// TIA Portal V17 export
// export: Created 2025-03-07T09:24:28.1169824Z, ExportSetting WithDefaults, DisplayName Totally Integrated Automation Portal, DisplayVersion V17 Update 8, DisplayName TIA Portal Openness, DisplayVersion V17 Update 8, DisplayName TIA Portal Version Control Interface, DisplayVersion V17, DisplayName SINAMICS Startdrive Advanced, DisplayVersion V17 SP2, DisplayName SINAMICS Startdrive G110M, G120, G120C, G120D, G120P, G115D, DisplayVersion V17 SP2, DisplayName SINAMICS Startdrive G130, G150, S120, S150, SINAMICS MV, S210, DisplayVersion V17 SP2, DisplayName STEP 7 Professional, DisplayVersion V17 Update 8, DisplayName SINUMERIK ONE STEP 7 Toolbox, DisplayVersion V17 Update 12, DisplayName SINUMERIK 840D sl STEP 7 Toolbox, DisplayVersion V17 Update 12, DisplayName STEP 7 Safety, DisplayVersion V17 Update 6, DisplayName WinCC Advanced, DisplayVersion V17 Update 8
FUNCTION_BLOCK "FB1015_E-STOP"   // FB1015, F_LAD
{ S7_Optimized_Access := 'TRUE' }
AUTHOR : ETXETAR
VERSION : 1.0
// stored: AutoNumber false, IsIECCheckEnabled false, UDAEnableTagReadback false
   VAR_INPUT
      SAFETY_DOORS_BYPASS : Bool;   // MACHINE SAFETY DOORS BYPASS IN EMERGENCY RESET INPUT
      FEEDBACK_OFF_E_STOP_IN : Bool;   // FEEDBACK OFF E-STOP INPUT
      FEEDBACK_OFF_E_STOP_RST_STR_IN : Bool;   // FEEDBACK OFF E-STOP RESET START INPUT
      MACH_E_STOP : Bool;   // MACHINE E-STOP INPUT
      POWDER_E_STOP : Bool;   // GANTRY E-STOP INPUT
   END_VAR
   VAR_OUTPUT
      E_STOP_OK : Bool;   // E-STOP OK OUTPUT
      E_STOP_OK_OFF_DEL_2 : Bool;   // E-STOP OK DELAYED 2 OUTPUT
      E_STOP_OK_OFF_DEL_3 : Bool;   // E-STOP OK DELAYED 3 OUTPUT
      E_STOP_OK_OFF_DEL_4 : Bool;   // E-STOP OK DELAYED 4 OUTPUT
      FEEDBACK_ERROR : Bool;   // E-STOP OK FEEDBACK ERROR
   END_VAR
   VAR
      ALL_E_STOP_IN : Bool;   // ALL E-STOP INPUTS
      E_STOP_RESET : Bool;   // E-STOP RESET
      E_STOP_RESET_REQ : Bool;   // E-STOP RESET REQUEST
      FEEDBACK_OFF_OK : Bool;   // E-STOP FEEDBACK OFF OK
      ESTOP1_Instance : ESTOP1;
      F_IEC_Timer_Instance : TOF;
      F_IEC_Timer_Instance_1 : TOF;
      F_IEC_TIMER_FBCK_OK : TON;
      F_IEC_Timer_Instance_2 : TOF;
   END_VAR
   VAR CONSTANT
      FB_NUMBER : DInt := 1014;
   END_VAR
   // F_IEC_TIMER_FBCK_OK.PT := T#30ms;
BEGIN

REGION Network 1: ALL EMERGENCY STOP INPUTS
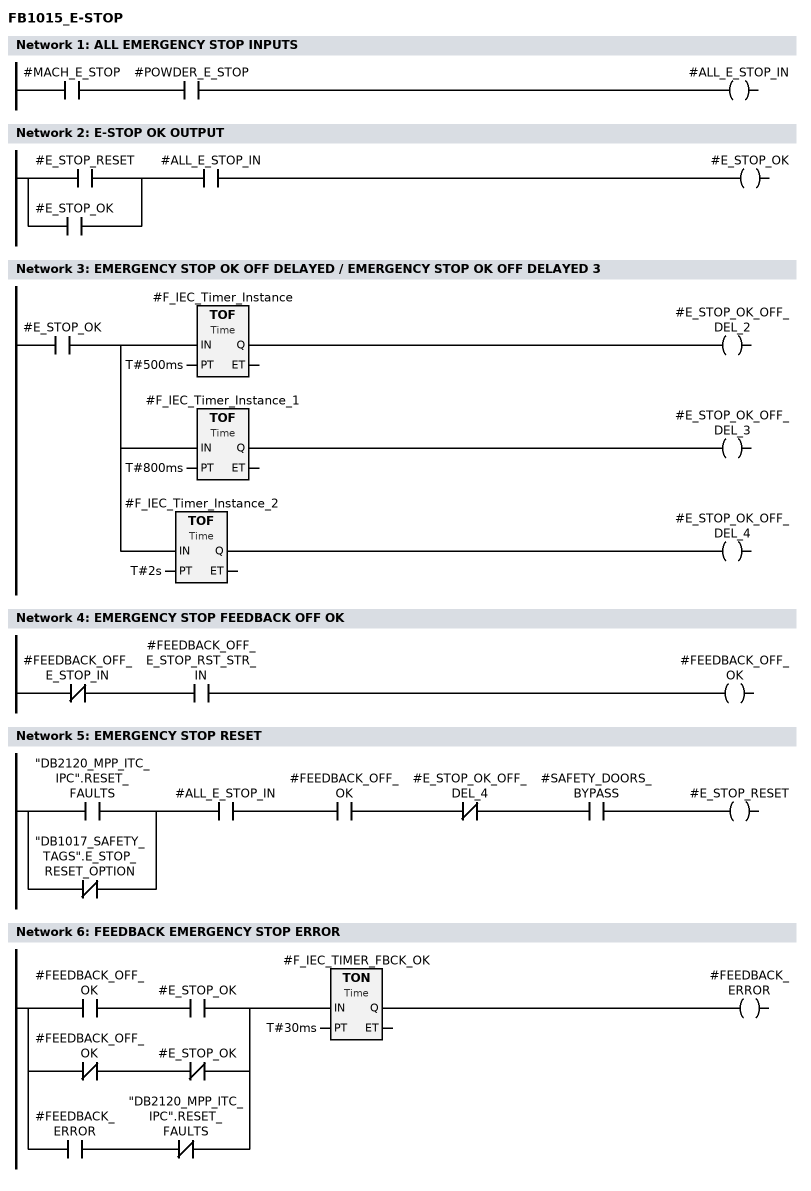
   RUNG wire#powerrail
      Contact( #MACH_E_STOP )
      Contact( #POWDER_E_STOP )
      Coil( #ALL_E_STOP_IN )
   END_RUNG
   // the same network as SCL:
   #ALL_E_STOP_IN := #MACH_E_STOP AND #POWDER_E_STOP;
END_REGION

REGION Network 2: E-STOP OK OUTPUT
   RUNG wire#powerrail
      Contact( #E_STOP_RESET )
      wire#w1
      Contact( #ALL_E_STOP_IN )
      Coil( #E_STOP_OK )
   END_RUNG
   RUNG wire#powerrail
      Contact( #E_STOP_OK )
   END_RUNG wire#w1
   // the same network as SCL:
   #E_STOP_OK := (#E_STOP_RESET OR #E_STOP_OK) AND #ALL_E_STOP_IN;
END_REGION

REGION Network 3: EMERGENCY STOP OK OFF DELAYED / EMERGENCY STOP OK OFF DELAYED 3
   RUNG wire#powerrail
      Contact( #E_STOP_OK )
      wire#w1
      { S7_Templates := "[time_type := Time, codedbool_type := DInt]" } #F_IEC_Timer_Instance.TOF(pt := T#500ms, et =>)
      Coil( #E_STOP_OK_OFF_DEL_2 )
   END_RUNG
   RUNG wire#w1
      { S7_Templates := "[time_type := Time, codedbool_type := DInt]" } #F_IEC_Timer_Instance_1.TOF(pt := T#800ms, et =>)
      Coil( #E_STOP_OK_OFF_DEL_3 )
   END_RUNG
   RUNG wire#w1
      { S7_Templates := "[time_type := Time, codedbool_type := DInt]" } #F_IEC_Timer_Instance_2.TOF(pt := T#2s, et =>)
      Coil( #E_STOP_OK_OFF_DEL_4 )
   END_RUNG
   // the same network as SCL:
   #F_IEC_Timer_Instance.TOF(IN := #E_STOP_OK, PT := T#500ms);
   #E_STOP_OK_OFF_DEL_2 := #F_IEC_Timer_Instance.Q;
   #F_IEC_Timer_Instance_1.TOF(IN := #E_STOP_OK, PT := T#800ms);
   #E_STOP_OK_OFF_DEL_3 := #F_IEC_Timer_Instance_1.Q;
   #F_IEC_Timer_Instance_2.TOF(IN := #E_STOP_OK, PT := T#2s);
   #E_STOP_OK_OFF_DEL_4 := #F_IEC_Timer_Instance_2.Q;
END_REGION

REGION Network 4: EMERGENCY STOP FEEDBACK OFF OK
   RUNG wire#powerrail
      I_Contact( #FEEDBACK_OFF_E_STOP_IN )
      Contact( #FEEDBACK_OFF_E_STOP_RST_STR_IN )
      Coil( #FEEDBACK_OFF_OK )
   END_RUNG
   // the same network as SCL:
   #FEEDBACK_OFF_OK := NOT #FEEDBACK_OFF_E_STOP_IN AND #FEEDBACK_OFF_E_STOP_RST_STR_IN;
END_REGION

REGION Network 5: EMERGENCY STOP RESET
   RUNG wire#powerrail
      Contact( "DB2120_MPP_ITC_IPC".RESET_FAULTS )
      wire#w1
      Contact( #ALL_E_STOP_IN )
      Contact( #FEEDBACK_OFF_OK )
      I_Contact( #E_STOP_OK_OFF_DEL_4 )
      Contact( #SAFETY_DOORS_BYPASS )
      Coil( #E_STOP_RESET )
   END_RUNG
   RUNG wire#powerrail
      I_Contact( "DB1017_SAFETY_TAGS".E_STOP_RESET_OPTION )
   END_RUNG wire#w1
   // the same network as SCL:
   #E_STOP_RESET := ("DB2120_MPP_ITC_IPC".RESET_FAULTS OR NOT "DB1017_SAFETY_TAGS".E_STOP_RESET_OPTION) AND #ALL_E_STOP_IN AND #FEEDBACK_OFF_OK AND NOT #E_STOP_OK_OFF_DEL_4 AND #SAFETY_DOORS_BYPASS;
END_REGION

REGION Network 6: FEEDBACK EMERGENCY STOP ERROR
   RUNG wire#powerrail
      Contact( #FEEDBACK_OFF_OK )
      Contact( #E_STOP_OK )
      wire#w1
      { S7_Templates := "[time_type := Time, codedbool_type := DInt]" } #F_IEC_TIMER_FBCK_OK.TON(pt := T#30ms, et =>)
      Coil( #FEEDBACK_ERROR )
   END_RUNG
   RUNG wire#powerrail
      I_Contact( #FEEDBACK_OFF_OK )
      I_Contact( #E_STOP_OK )
   END_RUNG wire#w1
   RUNG wire#powerrail
      Contact( #FEEDBACK_ERROR )
      I_Contact( "DB2120_MPP_ITC_IPC".RESET_FAULTS )
   END_RUNG wire#w1
   // the same network as SCL:
   #F_IEC_TIMER_FBCK_OK.TON(IN := (#FEEDBACK_OFF_OK AND #E_STOP_OK) OR (NOT #FEEDBACK_OFF_OK AND NOT #E_STOP_OK) OR (#FEEDBACK_ERROR AND NOT "DB2120_MPP_ITC_IPC".RESET_FAULTS),
                           PT := T#30ms);
   #FEEDBACK_ERROR := #F_IEC_TIMER_FBCK_OK.Q;
END_REGION
END_FUNCTION_BLOCK
